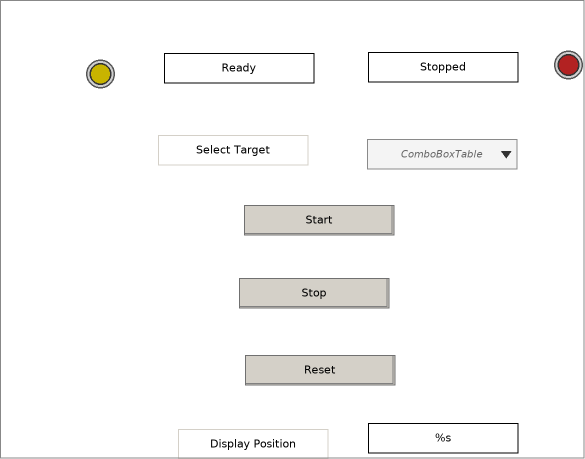
VISUALIZATION Control_HMI  // 585x459
    Textfield (158,135 150x30), "Select Target"
    Rectangle (368,423 150x30), "%s", text variable: GVL.qxDIsplay_Pos
    Textfield (178,429 150x30), "Display Position"
    Button (244,205 150x30), "Start"
        tap GVL.ixStartButton
    Button (239,278 150x30), "Stop"
        tap GVL.ixStopButton
    Button (245,355 150x30), "Reset"
        tap GVL.ixResetButton
    Lamp1 (84,57 33x34), variable: GVL.qxReadylamp, style: Lamp-Lamp1-Yellow
    Lamp1 (552,48 33x34), variable: GVL.qxStoplamp, style: Lamp-Lamp1-Red
    ComboBoxTable (367,139 150x30), variable: GVL.Position, data array: GVL.sTargetList
        p3854506369: GVL.sTargetList[INDEX]
    RoundedRectangle (164,53 150x30), "Ready"
    RoundedRectangle (368,52 150x30), "Stopped"
END_VISUALIZATION

(* stored: Version 1.1.0.1, ProductVersion 3.1.4024.12
   Visu Control_HMI: Id {1e57c2b1-51d9-479f-8f1d-f3b2fdb20f9a} *)
